# EPICS IOC start-up script: commonIocsh/iocsh/linStatHost.iocsh
#--################################################################################################
#--############### START of linStatHost.iocsh #####################################################
#-- IOC     : Record name prefix
#-- LINSTAT : linStat module install top (db under $(LINSTAT)/db)
#--################################################################################################
#--#
#--# Host-wide Linux system statistics: memory, CPU, uptime, hwmon, IRQ.
#--# Load before iocInit. Loaded by default from the global linStat.iocsh.
#--#
#--# Do not load together with iocStatsAdmin.iocsh for the same IOC: both create records of the
#--# same names, and the second load fails.
#--#
#-
dbLoadRecords("$(LINSTAT)/db/linStatHost.db", "IOC=$(IOC)")
#-
#--############### END of linStatHost.iocsh #######################################################
#--################################################################################################
